(* CODESYS project Daramic_FINAL_MC2_TM218LDA24DRN_05_01_19.project
   Title: Daramic_Cutting
   Version: 0.0.0.40

Project tree, tasks and I/O mapping:
  MyController : TM218LDA24DRN, Schneider Electric, order no. TM218LDA24DRN, version 4.0.1.26
      settings: Expansion Tasks.Expansion 1 Task Name = 'MAST'; Expansion Tasks.Expansion 2 Task Name = 'MAST'
    application Application
      libraries: Standard, * (System)
      task MAST (cyclic, interval 20 ms, priority 15, watchdog 100 ms x 1) calls MainPOU
      global variables GVL
      program MainPOU [FBD]
      function block cutterPID [ST]
      trace Trace (task MAST): MPM, MainPOU.initSetCutRPM, MainPOU.midSetCutRPM, MainPOU.laterSetCutRPM2, MainPOU.laterSetCutRPM, MainPOU.finalSetCutRPM
      function block RPMtimer [ST]
      function block MPMAveraging [ST]
      function HiddenPOU [ST]
    Serial Line 1
      SoMachine_Network_Manager : SoMachine-Network Manager, Schneider Electric, version 4.0.0.2
    Serial Line 2
      Modbus_Manager : Modbus Manager, Schneider Electric, version 4.0.0.2
    Embedded Functions
      IO : IO, Schneider Electric, version 4.0.1.26
          input  iCountingSensor : BOOL  // IW0.I1
          input  iStartPB : BOOL  // IW0.I4
          input  iEStop : BOOL  // IW0.I5
          input  iAutoSleeving : BOOL  // IW0.I6
          input  iFootSwitch : BOOL  // IW0.I7
          input  iPhotoMatDetect : BOOL  // IW0.I8
          input  iUnwindingSensor : BOOL  // IW0.I9
          input  iDoorLS : BOOL  // IW0.I10
          input  iPhotoConv : BOOL  // IW0.I11
          input  iInching : BOOL  // IW0.I12
          input  iStopPB : BOOL  // IW0.I13
          output qStartFeeding : BOOL  // QW0.Q0
          output qStartCutting : BOOL  // QW0.Q1
          output qStartSleeve : BOOL  // QW0.Q3
          output qLightGreen : BOOL  // QW0.Q6
          output qLightYellow : BOOL  // QW0.Q7
          output qLightRed : BOOL  // QW0.Q8
          output qInterlock : BOOL  // QW0.Q9
          unmapped channels: IW0, QW0
      HSC : HSC, Schneider Electric, version 4.0.1.26
          settings: HSC00VarName = ''; HSC01VarName = ''
    Module_5 : TM2AMO1HT, Schneider Electric, order no. TM2AMO1HT, version 4.0.1.26
        settings: QW0.Maximum = 2800
        output qwSealingRPM : INT  // QW0
    Module_4 : TM2AMO2HTN, Schneider Electric, order no. TM2AMO2HTN, version 4.0.1.26
        settings: QW0.Maximum = 2800; QW1.Maximum = 2800
        output qwFeedRPM : INT  // QW0
        output qwCutterRPM : INT  // QW1
*)

// MyController/Application/GVL
VAR_GLOBAL
	// REAL: MD0 to MD49 (MW0 to MW98)
	// INT: MW100 to MW199
	// BOOL: MX400 to MX598 (MW200 to MW299)
	MPM : REAL;
	displayMPM AT %MD6: REAL;
	convMPM AT %MD7: REAL;
	actualCutLength AT %MD8: REAL;
	
	countReset AT %MX400.0: BOOL;
	enableCorrection AT %MX400.1: BOOL;
	countStart AT %MX400.2: BOOL;
	countEnabled AT %MX400.3: BOOL;
	iStart: BOOL;
	setCutLength: REAL := 100;
	
END_VAR

VAR_GLOBAL RETAIN
	feedRollDia AT %MD0: REAL := 76.5;
	conveyorRollDia AT %MD1: REAL := 76.5;
	setCutLength1 AT %MD2: REAL := 200;
	setMPM AT %MD3: REAL;
	lengthTolerance AT %MD4: REAL := 0.5;
	offsetLength AT %MD5 : REAL;
	offsetRPM: REAL;
	cutCount AT %MW100: INT;
	cutCountRetain: DWORD;
	cutCountRetainWord: WORD;
	sealingRatio AT %MD10 : REAL := 1.67;
	offsetOperator AT %MD9: REAL;
END_VAR

// MyController/Application/MainPOU
PROGRAM MainPOU
VAR
	feedEncoderVal: DINT;
	convEncoderVal: DINT;
	feedRPM: REAL;
	setFeedRPM: REAL;
	setCutRPM: REAL;
	convRPM: REAL;
	TON_0: TON;
	timerET: TIME;
	timerETINT: INT;
	timeMatDetect: INT;
	F_TRIG_0: F_TRIG;
	MatDetectTime: INT;
	CTU_0: CTU;
	R_TRIG_0: R_TRIG;
	cutterPID_0: cutterPID;
	R_TRIG_1: R_TRIG;
	RS_0: RS;
	initSetCutRPM: REAL;
	TON_1: TON;
	laterSetCutRPM: REAL;
	startFeedDelay: BOOL;
	TON_2: TON;
	actCutterRPM: REAL;
	PID_0: PID;
	setCutRPM1: REAL;
	setCutRPMPID: REAL;
	TON_3: TON;
	TON_4: TON;
	startFeedingDelay: BOOL;
	TON_5: TON;
	midSetCutRPM: REAL;
	setCutRPM2: REAL;
	aa: REAL;
	scutrpmet: INT;
	finalSetCutRPM: REAL;
	laterSetCutRPM2: REAL;
	setCutRPM3: REAL;
	setCutRPM4: REAL;
	TON_6: TON;
	TON_7: TON;
	setCutRPM5: REAL;
	RPMtimer_0: RPMtimer;
	TON_8: TON;
	mcRunning: BOOL;
	RPMtimer_1: RPMtimer;
	MPMavg: REAL;
	MPMAveraging_0: MPMAveraging;
	counterre: BOOL;
	cutCountDWORD: DWORD;
	cutCountWORD: WORD;
	hscRunFB: BOOL;
	HSCSetParam_0: HSCSetParam;
	setCurrValDone: BOOL;
	RS_1: RS;
	sr1: SR;
	hscWasOff: BOOL;
	SR_0: SR;
	resetMaintained: BOOL;
	TON_9: TON;
	TON_10: TON;
	TON_11: TON;
	CTUD_0: CTUD;
	resetCtud: BOOL;
	TON_12: TON;
	TON_13: TON;
END_VAR
VAR // added by the converter: edge detectors and wires of the graphical bodies
    _w1, _w2 : BOOL;
END_VAR

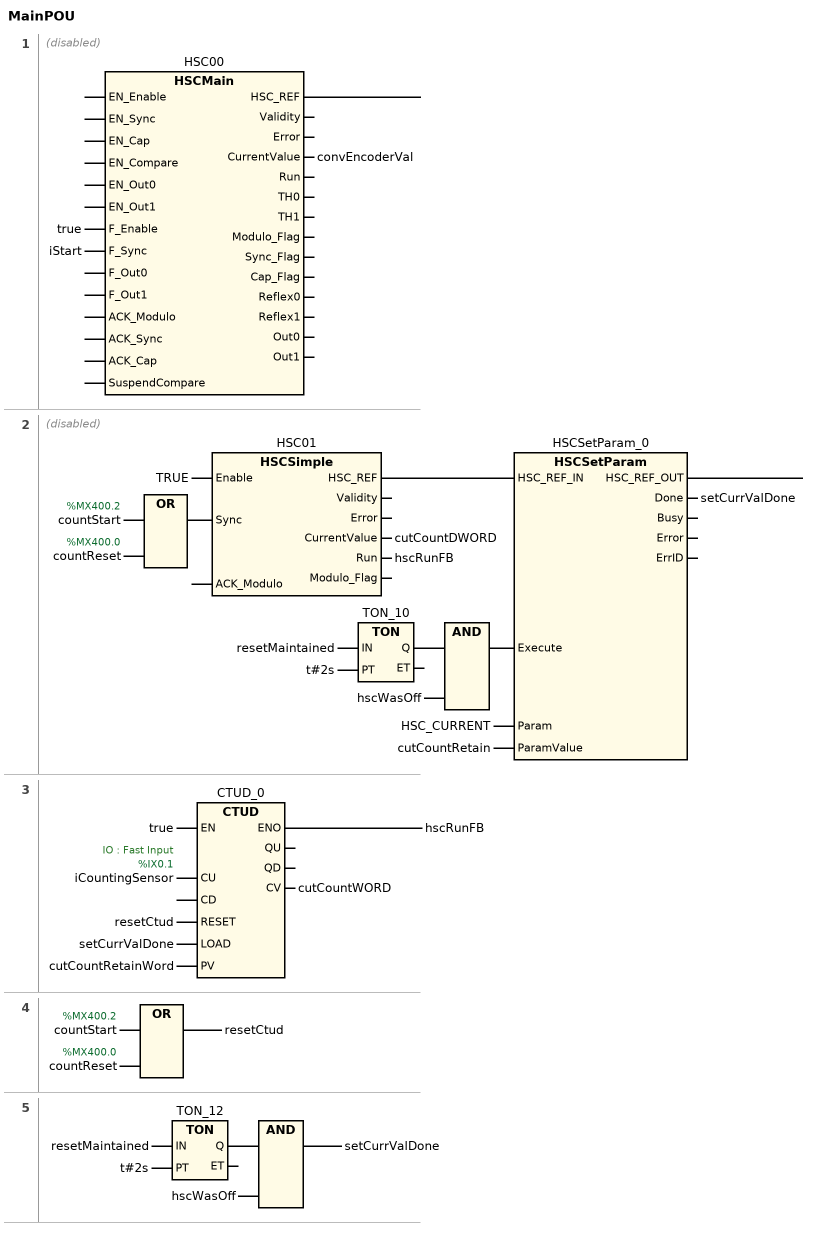
// NETWORK 1 (disabled)
// HSC00(F_Enable := true, F_Sync := iStart, CurrentValue => convEncoderVal); // HSCMain

// NETWORK 2 (disabled)
//   countStart: AT %MX400.2
//   countReset: AT %MX400.0
// HSC01(Enable := TRUE, Sync := countStart OR countReset, CurrentValue => cutCountDWORD, Run => hscRunFB); // HSCSimple
// TON_10(IN := resetMaintained, PT := t#2s); // TON
// HSCSetParam_0(
//     HSC_REF_IN := HSC01.HSC_REF,
//     Execute := TON_10.Q AND hscWasOff,
//     Param := HSC_CURRENT,
//     ParamValue := cutCountRetain,
//     Done => setCurrValDone); // HSCSetParam

// NETWORK 3
//   iCountingSensor: IO : Fast Input | AT %IX0.1
_w1 := true;
IF _w1 THEN
    CTUD_0(
        CU := iCountingSensor,
        RESET := resetCtud,
        LOAD := setCurrValDone,
        PV := cutCountRetainWord,
        CV => cutCountWORD); // CTUD
END_IF
hscRunFB := _w1;

// NETWORK 4
//   countStart: AT %MX400.2
//   countReset: AT %MX400.0
resetCtud := countStart OR countReset;

// NETWORK 5
TON_12(IN := resetMaintained, PT := t#2s); // TON
setCurrValDone := TON_12.Q AND hscWasOff;

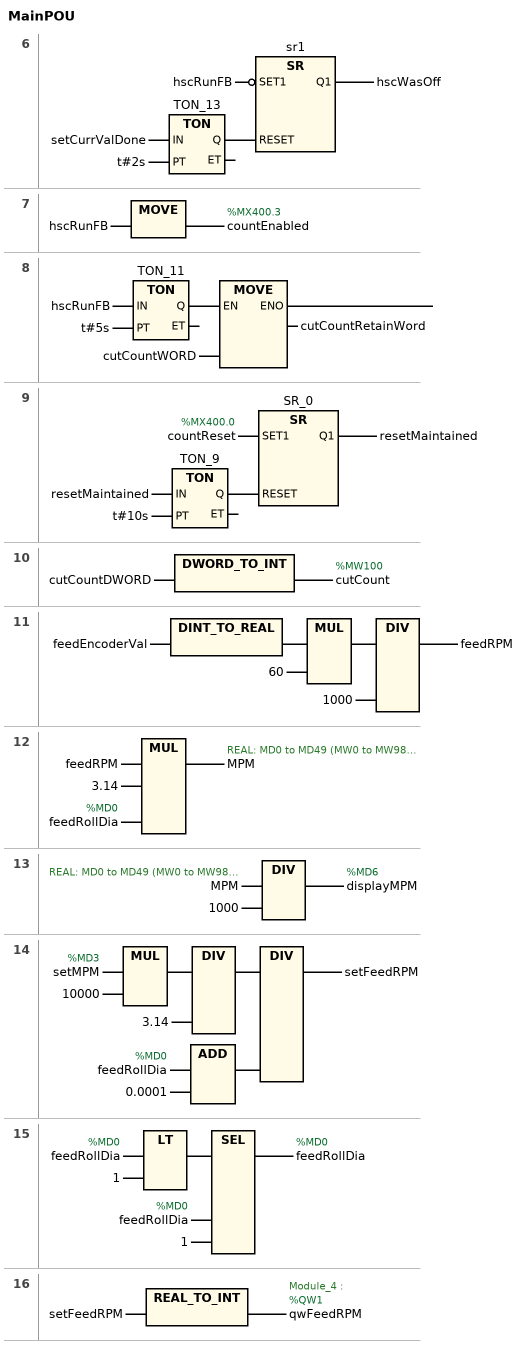
// NETWORK 6
TON_13(IN := setCurrValDone, PT := t#2s); // TON
sr1(SET1 := NOT hscRunFB, RESET := TON_13.Q); // SR
hscWasOff := sr1.Q1;

// NETWORK 7
//   countEnabled: AT %MX400.3
countEnabled := hscRunFB;

// NETWORK 8
TON_11(IN := hscRunFB, PT := t#5s); // TON
IF TON_11.Q THEN cutCountRetainWord := cutCountWORD; END_IF

// NETWORK 9
//   countReset: AT %MX400.0
TON_9(IN := resetMaintained, PT := t#10s); // TON
SR_0(SET1 := countReset, RESET := TON_9.Q); // SR
resetMaintained := SR_0.Q1;

// NETWORK 10
//   cutCount: AT %MW100
cutCount := DWORD_TO_INT(cutCountDWORD);

// NETWORK 11
feedRPM := (DINT_TO_REAL(feedEncoderVal) * 60) / 1000;

// NETWORK 12
//   feedRollDia: AT %MD0
//   MPM: REAL: MD0 to MD49 (MW0 to MW98) INT: MW100 to MW199 BOOL: MX400 to MX598 (MW200 to MW299)
MPM := feedRPM * 3.14 * feedRollDia;

// NETWORK 13
//   MPM: REAL: MD0 to MD49 (MW0 to MW98) INT: MW100 to MW199 BOOL: MX400 to MX598 (MW200 to MW299)
//   displayMPM: AT %MD6
displayMPM := MPM / 1000;

// NETWORK 14
//   setMPM: AT %MD3
//   feedRollDia: AT %MD0
setFeedRPM := ((setMPM * 10000) / 3.14) / (feedRollDia + 0.0001);

// NETWORK 15
//   feedRollDia: AT %MD0
feedRollDia := SEL(feedRollDia < 1, feedRollDia, 1);

// NETWORK 16
//   qwFeedRPM: Module_4 : | AT %QW1
qwFeedRPM := REAL_TO_INT(setFeedRPM);

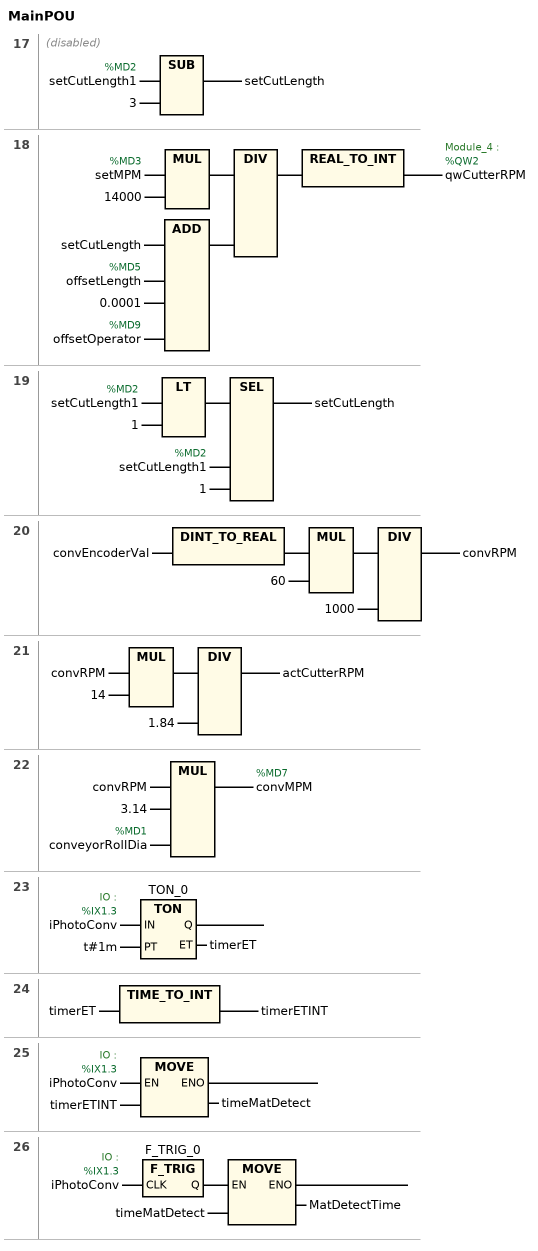
// NETWORK 17 (disabled)
//   setCutLength1: AT %MD2
// setCutLength := setCutLength1 - 3;

// NETWORK 18
//   setMPM: AT %MD3
//   offsetLength: AT %MD5
//   offsetOperator: AT %MD9
//   qwCutterRPM: Module_4 : | AT %QW2
qwCutterRPM := REAL_TO_INT((setMPM * 14000) / (setCutLength + offsetLength + 0.0001 + offsetOperator));

// NETWORK 19
//   setCutLength1: AT %MD2
setCutLength := SEL(setCutLength1 < 1, setCutLength1, 1);

// NETWORK 20
convRPM := (DINT_TO_REAL(convEncoderVal) * 60) / 1000;

// NETWORK 21
actCutterRPM := (convRPM * 14) / 1.84;

// NETWORK 22
//   conveyorRollDia: AT %MD1
//   convMPM: AT %MD7
convMPM := convRPM * 3.14 * conveyorRollDia;

// NETWORK 23
//   iPhotoConv: IO : | AT %IX1.3
TON_0(IN := iPhotoConv, PT := t#1m, ET => timerET); // TON

// NETWORK 24
timerETINT := TIME_TO_INT(timerET);

// NETWORK 25
//   iPhotoConv: IO : | AT %IX1.3
IF iPhotoConv THEN timeMatDetect := timerETINT; END_IF

// NETWORK 26
//   iPhotoConv: IO : | AT %IX1.3
F_TRIG_0(CLK := iPhotoConv); // F_TRIG
IF F_TRIG_0.Q THEN MatDetectTime := timeMatDetect; END_IF

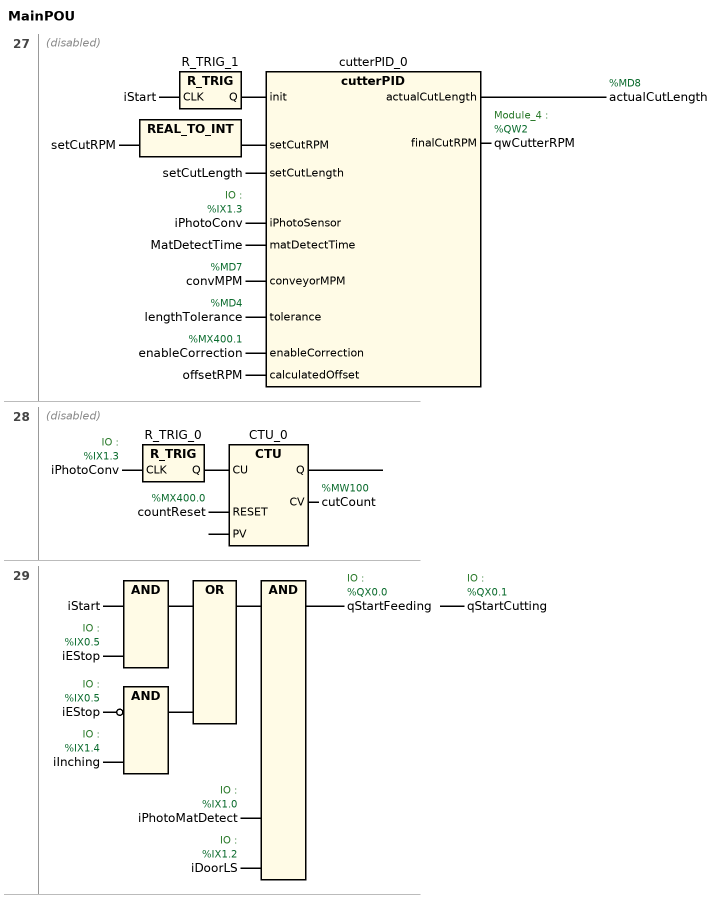
// NETWORK 27 (disabled)
//   iPhotoConv: IO : | AT %IX1.3
//   convMPM: AT %MD7
//   lengthTolerance: AT %MD4
//   enableCorrection: AT %MX400.1
//   qwCutterRPM: Module_4 : | AT %QW2
//   actualCutLength: AT %MD8
// R_TRIG_1(CLK := iStart); // R_TRIG
// cutterPID_0(
//     init := R_TRIG_1.Q,
//     setCutRPM := REAL_TO_INT(setCutRPM),
//     setCutLength := setCutLength,
//     iPhotoSensor := iPhotoConv,
//     matDetectTime := MatDetectTime,
//     conveyorMPM := convMPM,
//     tolerance := lengthTolerance,
//     enableCorrection := enableCorrection,
//     calculatedOffset := offsetRPM,
//     finalCutRPM => qwCutterRPM); // cutterPID
// actualCutLength := cutterPID_0.actualCutLength;

// NETWORK 28 (disabled)
//   iPhotoConv: IO : | AT %IX1.3
//   countReset: AT %MX400.0
//   cutCount: AT %MW100
// R_TRIG_0(CLK := iPhotoConv); // R_TRIG
// CTU_0(CU := R_TRIG_0.Q, RESET := countReset, CV => cutCount); // CTU

// NETWORK 29
//   iEStop: IO : | AT %IX0.5
//   iInching: IO : | AT %IX1.4
//   iPhotoMatDetect: IO : | AT %IX1.0
//   iDoorLS: IO : | AT %IX1.2
//   qStartFeeding: IO : | AT %QX0.0
//   qStartCutting: IO : | AT %QX0.1
_w2 := (iStart AND iEStop OR NOT iEStop AND iInching) AND iPhotoMatDetect AND iDoorLS;
qStartFeeding := _w2;
qStartCutting := _w2;

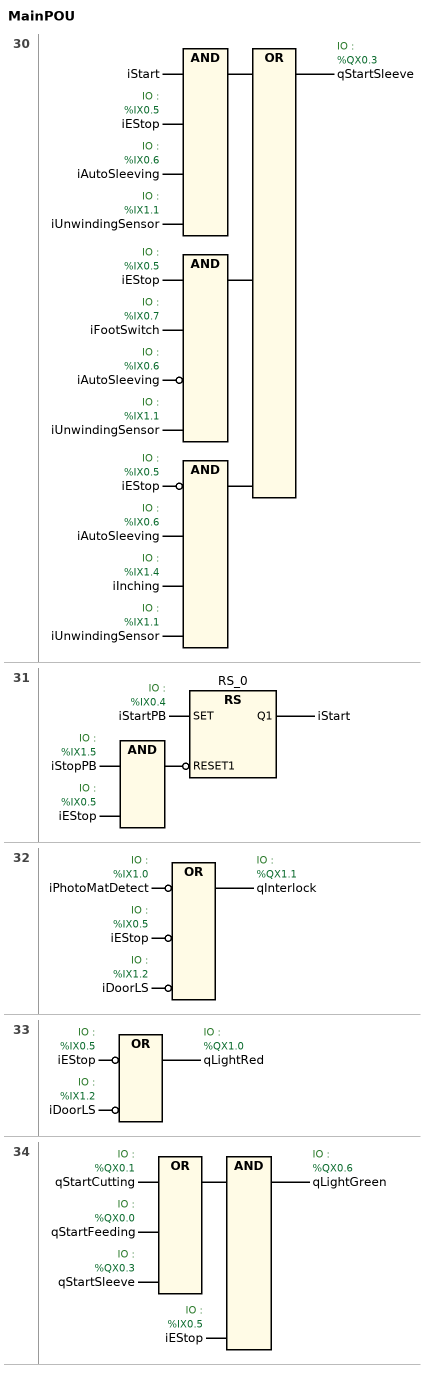
// NETWORK 30
//   iEStop: IO : | AT %IX0.5
//   iAutoSleeving: IO : | AT %IX0.6
//   iUnwindingSensor: IO : | AT %IX1.1
//   iFootSwitch: IO : | AT %IX0.7
//   iInching: IO : | AT %IX1.4
//   qStartSleeve: IO : | AT %QX0.3
qStartSleeve := iStart AND iEStop AND iAutoSleeving AND iUnwindingSensor OR iEStop AND iFootSwitch AND NOT iAutoSleeving AND iUnwindingSensor OR NOT iEStop AND iAutoSleeving AND iInching AND iUnwindingSensor;

// NETWORK 31
//   iStartPB: IO : | AT %IX0.4
//   iStopPB: IO : | AT %IX1.5
//   iEStop: IO : | AT %IX0.5
RS_0(SET := iStartPB, RESET1 := NOT (iStopPB AND iEStop)); // RS
iStart := RS_0.Q1;

// NETWORK 32
//   iPhotoMatDetect: IO : | AT %IX1.0
//   iEStop: IO : | AT %IX0.5
//   iDoorLS: IO : | AT %IX1.2
//   qInterlock: IO : | AT %QX1.1
qInterlock := NOT iPhotoMatDetect OR NOT iEStop OR NOT iDoorLS;

// NETWORK 33
//   iEStop: IO : | AT %IX0.5
//   iDoorLS: IO : | AT %IX1.2
//   qLightRed: IO : | AT %QX1.0
qLightRed := NOT iEStop OR NOT iDoorLS;

// NETWORK 34
//   qStartCutting: IO : | AT %QX0.1
//   qStartFeeding: IO : | AT %QX0.0
//   qStartSleeve: IO : | AT %QX0.3
//   iEStop: IO : | AT %IX0.5
//   qLightGreen: IO : | AT %QX0.6
qLightGreen := (qStartCutting OR qStartFeeding OR qStartSleeve) AND iEStop;

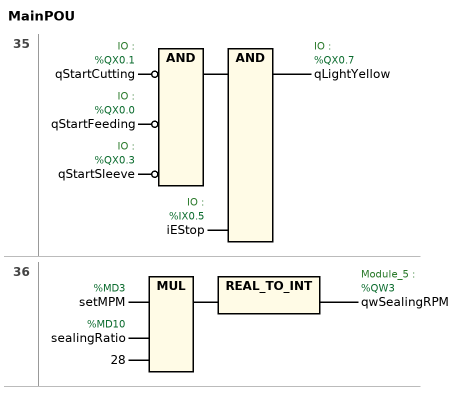
// NETWORK 35
//   qStartCutting: IO : | AT %QX0.1
//   qStartFeeding: IO : | AT %QX0.0
//   qStartSleeve: IO : | AT %QX0.3
//   iEStop: IO : | AT %IX0.5
//   qLightYellow: IO : | AT %QX0.7
qLightYellow := (NOT qStartCutting AND NOT qStartFeeding AND NOT qStartSleeve) AND iEStop;

// NETWORK 36
//   setMPM: AT %MD3
//   sealingRatio: AT %MD10
//   qwSealingRPM: Module_5 : | AT %QW3
qwSealingRPM := REAL_TO_INT(setMPM * sealingRatio * 28);

END_PROGRAM

// MyController/Application/cutterPID
FUNCTION_BLOCK cutterPID
VAR_INPUT
	init: BOOL;
	setCutRPM: INT;
	setCutLength: REAL;
	iPhotoSensor: BOOL;
	matDetectTime: INT;
	conveyorMPM: REAL;
	tolerance: REAL;
	enableCorrection: BOOL;
END_VAR
VAR_OUTPUT
	actualCutLength: REAL;
	finalCutRPM: INT;
	
END_VAR
VAR
	et1: INT :=0;
	et2: INT := 0;
	et3: INT :=0;
	et4: INT :=0;
	et5: INT :=0;
	totalET: INT :=0;
	ctu1: CTU;
	var1: BOOL;
END_VAR

VAR_IN_OUT
	calculatedOffset: REAL :=0;
END_VAR

IF init THEN
	et1 := 0;
	et2 := 0;
	et3 := 0;
	et4 := 0;
	et5 := 0;
END_IF
ctu1(CU:= iPhotoSensor, RESET:= var1, PV := 5);
var1:= ctu1.Q;
CASE  ctu1.CV OF
	1: et1 := matDetectTime;
	2: et2 := matDetectTime;
	3: et3 := matDetectTime;
	4: et4 := matDetectTime;
	5: et5 := matDetectTime;
END_CASE

IF et5 = 0 THEN
	actualCutLength := (conveyorMPM * ET1)/ (60*1000);
ELSE
totalET := et1+et2+et3+et4+et5;
actualCutLength := (conveyorMPM * totalET)/ (5*60*1000);
END_IF
IF enableCorrection THEN
	IF actualCutLength > (setCutLength + tolerance) THEN
		finalCutRPM := setCutRPM + 1;
	ELSIF actualCutLength < (setCutLength - tolerance) THEN
		finalCutRPM := setCutRPM - 1;
	END_IF
	calculatedOffset := finalCutRPM - setCutRPM;
ELSE
	finalCutRPM := setCutRPM;
END_IF

END_FUNCTION_BLOCK

// MyController/Application/RPMtimer
FUNCTION_BLOCK RPMtimer
VAR_INPUT
	enable: BOOL;
	inRPM: REAL; 
END_VAR
VAR_OUTPUT
	outRPM: REAL;
END_VAR
VAR
	
	var1: REAL := 0;
	var2: REAL := 0;
	var3: REAL := 0;
	var4: REAL := 0;
	var5: REAL := 0;
	ctu1: Standard.CTU;
	blink1: Util.BLINK;
	resetCounter: BOOL;
	num1: INT;
	num2: INT;
	num3: INT;
	num4: INT;
	num5: INT;
	totalnum: INT;
	total: INT;
END_VAR

IF enable THEN
	blink1(enable:= TRUE, timelow:= T#100MS, timehigh:= T#100MS);
	ctu1(cu:=blink1.OUT, reset:=resetCounter, pv:= 3);
	resetCounter := ctu1.Q;
	CASE ctu1.CV OF
	1:	var1 := inRPM;
	2:	var2 := inRPM;
	3:	var3 := inRPM;
	
	ELSE
		outRPM := inRPM;
	END_CASE
	IF var1 > 0 THEN
		num1 := 1;
	ELSE
		num1 := 0;
	END_IF
	IF var2 > 0 THEN
		num2 := 1;
	ELSE
		num2 := 0;
	END_IF
	IF var3 > 0 THEN
		num3 := 1;
	ELSE
		num3 := 0;
	END_IF
	
	totalnum := num1+num2+num3;
	IF totalnum = 0 THEN
		total := 1;
	ELSE
		total := totalnum;
	END_IF
	
	outRPM := (var1+var2+var3)/(total+0.0001);
ELSE
	outRPM := inRPM;
	var1:=0;
	var2:=0;
	var3:=0;
	var4:=0;
	var5:=0;
END_IF

END_FUNCTION_BLOCK

// MyController/Application/MPMAveraging
FUNCTION_BLOCK MPMAveraging
VAR_INPUT
	enable: BOOL;
	inputMPM: REAL; 
END_VAR
VAR_OUTPUT
	outMPM: REAL;
END_VAR
VAR
	t1: TON;
	var1: REAL := 0;
	var2: REAL := 0;
	var3: REAL := 0;
	var4: REAL := 0;
	var5: REAL := 0;
	var6: REAL := 0;
	var7: REAL := 0;
	var8: REAL := 0;
	var9: REAL := 0;
	var10: REAL := 0;
	ctu1: Standard.CTU;
	blink1: Util.BLINK;
	resetCounter: BOOL;
	num1: INT;
	num2: INT;
	num3: INT;
	num4: INT;
	num5: INT;
	num6: INT;
	num7: INT;
	num8: INT;
	num9: INT;
	num10: INT;
	totalnum: INT;
	total: INT;
	inMPM: REAL;
END_VAR

IF enable THEN
	t1(IN:=qStartFeeding, pt:=T#20S);
	IF t1.Q THEN
		IF inputMPM < (outMPM-25) THEN
			inMPM := outMPM - 15;
		ELSIF inputMPM > (outMPM+25) THEN
			inMPM := outMPM + 15;
		END_IF
	ELSE
		inMPM := inputMPM;
	END_IF
	
	blink1(enable:= TRUE, timelow:= T#100MS, timehigh:= T#100MS);
	ctu1(cu:=blink1.OUT, reset:=resetCounter, pv:= 10);
	resetCounter := ctu1.Q;
	CASE ctu1.CV OF
	1:	var1 := inMPM;
	2:	var2 := inMPM;
	3:	var3 := inMPM;
	4:	var4 := inMPM;
	5:	var5 := inMPM;
	6:	var6 := inMPM;
	7:	var7 := inMPM;
	8:	var8 := inMPM;
	9:	var9 := inMPM;
	10:	var10 := inMPM;
	ELSE
		outMPM := inMPM;
	END_CASE
	IF var1 > 0 THEN
		num1 := 1;
	ELSE
		num1 := 0;
	END_IF
	IF var2 > 0 THEN
		num2 := 1;
	ELSE
		num2 := 0;
	END_IF
	IF var3 > 0 THEN
		num3 := 1;
	ELSE
		num3 := 0;
	END_IF
	IF var4 > 0 THEN
		num4 := 1;
	ELSE
		num4 := 0;
	END_IF
	IF var5 > 0 THEN
		num5 := 1;
	ELSE
		num5 := 0;
	END_IF
	IF var6 > 0 THEN
		num6 := 1;
	ELSE
		num6 := 0;
	END_IF
	IF var7 > 0 THEN
		num7 := 1;
	ELSE
		num7 := 0;
	END_IF
	IF var8 > 0 THEN
		num8 := 1;
	ELSE
		num8 := 0;
	END_IF
	IF var9 > 0 THEN
		num9 := 1;
	ELSE
		num9 := 0;
	END_IF
	IF var10 > 0 THEN
		num10 := 1;
	ELSE
		num10 := 0;
	END_IF
	totalnum := num1+num2+num3+num4+num5+num6+num7+num8+num9+num10;
	IF totalnum = 0 THEN
		total := 1;
	ELSE
		total := totalnum;
	END_IF
	
	outMPM := (var1+var2+var3+var4+var5+var6+var7+var8+var9+var10)/(total+0.0001);
ELSE
	outMPM := inMPM;
	var1:=0;
	var2:=0;
	var3:=0;
	var4:=0;
	var5:=0;
	var6:=0;
	var7:=0;
	VAR8:=0;
	var9:=0;
	var10:=0;
END_IF

END_FUNCTION_BLOCK

// MyController/Application/HiddenPOU
FUNCTION HiddenPOU : BOOL

VAR_INPUT
	pHiddenFunc: POINTER TO WORD;
END_VAR
VAR
	pRead: POINTER TO BYTE;
	pWrite: POINTER TO BYTE;
END_VAR

pRead := pHiddenFunc + 400;
pWrite := pHiddenFunc + 4400;
HiddenPOU := TRUE;

END_FUNCTION
